{attribute 'linkalways'} 
{attribute 'no_explicit_call' := 'This FB is a CLASS and must be accessed using methods or properties'}
{attribute 'enable_dynamic_creation'}
FUNCTION_BLOCK Node_F_VN_MinElementElementwise_SINT EXTENDS VisionNode
VAR
    ipContainer : _ITcVnContainer;
    nMin : _SINT(0);
    hrPrev : _HRESULT(S_OK);
    hresult : _HRESULT(S_OK);
END_VAR

METHOD PUBLIC  Clone : I_Node
VAR
	pNode : POINTER TO Node_F_VN_MinElementElementwise_SINT;
END_VAR
pNode := __NEW(Node_F_VN_MinElementElementwise_SINT);
Clone := pNode^;
END_METHOD

METHOD FB_init : BOOL
VAR_INPUT
	bInitRetains : BOOL; // if TRUE, the retain variables are initialized (warm start / cold start)
	bInCopyCode : BOOL;  // if TRUE, the instance afterwards gets moved into the copy code (online change)
END_VAR
AddInput('ipContainer', ipContainer);
AddInput('nMin', nMin);
AddInput('hrPrev', hrPrev);
AddOutput('ipContainer', ipContainer);
AddOutput('hresult',hresult);
END_METHOD

METHOD PROTECTED OnExecute : HRESULT
hresult.Value := F_VN_MinElementElementwise_SINT(
    ipContainer := ipContainer.Value,
    nMin := nMin.Value,
    hrPrev:= hrPrev.Value);
END_METHOD

METHOD PUBLIC PreExecutionCheck
VAR_INPUT
	Check : I_PreExecutionChecks;
END_VAR
Check.IsTrue(ipContainer.IsValid, 'ipContainer must be a valid container');
Check.IsTrue(ipContainer.HasType(TC_GLOBAL_CONST_LIST.ContainerType_Vector_SINT), 'ipContainer contains incorrect type');
END_METHOD

END_FUNCTION_BLOCK

(* stored: Version 1.1.0.1, ProductVersion 3.1.4024.13
   POU Node_F_VN_MinElementElementwise_SINT: Id {a1143c28-d802-4e60-897c-634da9398216}, SpecialFunc None
   Folder Constructor: Id {932ab309-70c8-4f8b-85cc-8a7d4641d5c8}
   Method Clone: Id {0327be90-dbd7-4902-b052-bcadc4810330}
   Method FB_init: Id {d8dfa43b-a761-468d-a221-920917c91751}
   Method OnExecute: Id {81039ed1-6f4b-464c-88cb-acbae5318718}
   Method PreExecutionCheck: Id {9781def2-4f7e-4406-ae7f-79bde1790769} *)
